FUNCTION_BLOCK FB_Invokable
VAR
END_VAR

{attribute 'TcRpcEnable'}
METHOD Test : INT
VAR_IN_OUT
	Value :  INT;
	Value2 : INT;
END_VAR
Test 	:= Value * 2;
Value 	:= Test * 2;
Value2 	:= Value * 2;
END_METHOD

END_FUNCTION_BLOCK

(* stored: Version 1.1.0.1
   POU FB_Invokable: Id {74c5c950-f5d3-4656-9f37-c6756bb68b39}, SpecialFunc None
   Method Test: Id {4467b56b-83a1-447a-943e-2b6363167747} *)
